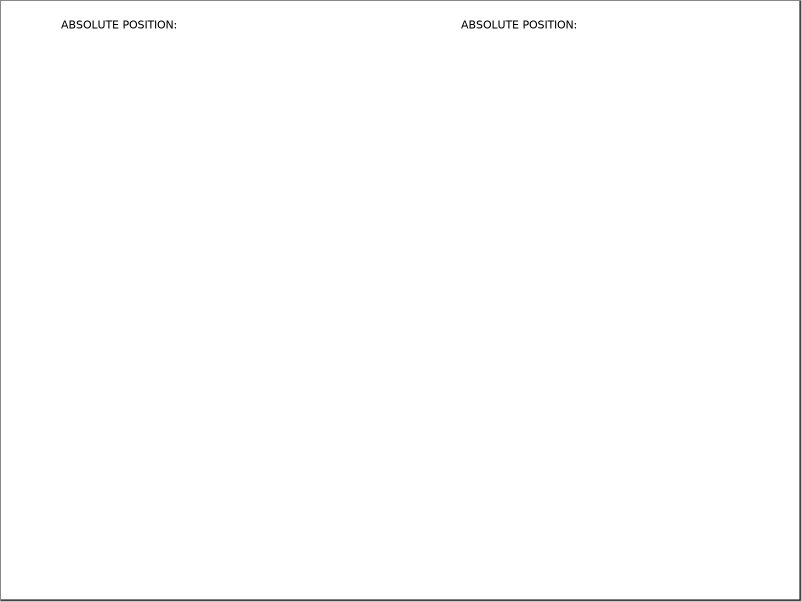
VISUALIZATION F12_Read_Actual_Position  // 802x602
    Rectangle (0,0 800x600)
    Label (10,10 170x30), "ABSOLUTE POSITION:"
    Label (410,10 170x30), "ABSOLUTE POSITION:"
END_VISUALIZATION

(* stored: Version 1.1.0.1, ProductVersion 3.1.4022.7
   Visu F12_Read_Actual_Position: Id {0e2ddf02-5a18-429a-93fe-d488251549aa} *)
